{attribute 'pack_mode=1'}
TYPE BR_to_TC_t :
STRUCT
END_STRUCT
END_TYPE

(* stored: Version 1.1.0.1, ProductVersion 3.1.4024.12
   DUT BR_to_TC_t: Id {8208c858-a7f5-46dc-a53e-0b037c467496} *)
